FUNCTION_BLOCK FB_WriteHPTSettings
VAR_INPUT
END_VAR
VAR_OUTPUT
END_VAR
VAR
	WriteSetting	: FB_WriteSDO;
	Step			: INT := 1;
	Debug1			: BOOL;
	DebugSize2		: BYTE;
	err				: BOOL;
	errId			: UDINT;
END_VAR

CASE Step OF

1:
// Write Thermocouple Ch1 settings
WriteSetting(
	nSlaveAddr := 1011,
	nIndex := 16#8000,
	nSubIndex := 16#01,
	bExecute := TRUE,
	nValueBool := 16#01
);

Debug1 := TO_BOOL(WriteSetting.nValueBool);

IF WriteSetting.bBusy = FALSE THEN
	Step := Step +1;
END_IF

2:
WriteSetting(
	nSlaveAddr := 1011,
	nIndex := 16#8000,
	nSubIndex := 16#07,
	nValueBool := 16#01,
	bExecute := TRUE
);

IF WriteSetting.bBusy = FALSE THEN
	Step := Step +1;
END_IF

3:
WriteSetting(
	nSlaveAddr := 1011,
	nIndex := 16#8000,
	nSubIndex := 16#08,
	nValueBool := 16#01,
	bExecute := TRUE
);

IF WriteSetting.bBusy = FALSE THEN
	Step := Step +1;
END_IF

4:
WriteSetting(
	nSlaveAddr := 1011,
	nIndex := 16#8000,
	nSubIndex := 16#12,
	nValueDInt := 31451,
	bExecute := TRUE
);

IF WriteSetting.bBusy = FALSE THEN
	Step := Step +1;
END_IF

5:
WriteSetting(
	nSlaveAddr := 1011,
	nIndex := 16#8000,
	nSubIndex := 16#13,
	nValueInt := -730,
	bExecute := TRUE
);

IF WriteSetting.bBusy = FALSE THEN
	Step := Step +1;
END_IF

6:
WriteSetting(
	nSlaveAddr := 1011,
	nIndex := 16#8000,
	nSubIndex := 16#14,
	nValueInt := 4820,
	bExecute := TRUE
);

IF WriteSetting.bBusy = FALSE THEN
	Step := Step +1;
END_IF

7:
// Write Thermocouple Ch2 settings
WriteSetting(
	nSlaveAddr := 1011,
	nIndex := 16#8010,
	nSubIndex := 16#01,
	nValueBool := 16#01,
	bExecute := TRUE
);

IF WriteSetting.bBusy = FALSE THEN
	Step := Step +1;
END_IF

8:
WriteSetting(
	nSlaveAddr := 1011,
	nIndex := 16#8010,
	nSubIndex := 16#07,
	nValueBool := 16#01,
	bExecute := TRUE
);

IF WriteSetting.bBusy = FALSE THEN
	Step := Step +1;
END_IF

9:
WriteSetting(
	nSlaveAddr := 1011,
	nIndex := 16#8010,
	nSubIndex := 16#08,
	nValueBool := 16#01,
	bExecute := TRUE
);

IF WriteSetting.bBusy = FALSE THEN
	Step := Step +1;
END_IF

10:
WriteSetting(
	nSlaveAddr := 1011,
	nIndex := 16#8010,
	nSubIndex := 16#12,
	nValueDInt := 31451,
	bExecute := TRUE
);

IF WriteSetting.bBusy = FALSE THEN
	Step := Step +1;
END_IF

11:
WriteSetting(
	nSlaveAddr := 1011,
	nIndex := 16#8010,
	nSubIndex := 16#13,
	nValueInt := -730,
	bExecute := TRUE
);

IF WriteSetting.bBusy = FALSE THEN
	Step := Step +1;
END_IF

12:
WriteSetting(
	nSlaveAddr := 1011,
	nIndex := 16#8010,
	nSubIndex := 16#14,
	nValueInt := 4820,
	bExecute := TRUE,
	bError => err,
	nErrId => errid
);

(*
// Write EL5042 encoder settings to enable correct readout
WriteSetting(
	nSlaveAddr := 1010,
	nIndex := 16#8008,
	nSubIndex := 16#15,
	nValue := 26,
	bExecute := TRUE
);

WriteSetting(
	nSlaveAddr := 1010,
	nIndex := 16#8008,
	nSubIndex := 16#16,
	nValue := 0,
	bExecute := TRUE
);

WriteSetting(
	nSlaveAddr := 1010,
	nIndex := 16#8018,
	nSubIndex := 16#15,
	nValue := 26,
	bExecute := TRUE
);

WriteSetting(
	nSlaveAddr := 1010,
	nIndex := 16#8018,
	nSubIndex := 16#16,
	nValue := 0,
	bExecute := TRUE
);
*)
Step := 1;
END_CASE

END_FUNCTION_BLOCK

(* stored: Version 1.1.0.1, ProductVersion 3.1.4024.2
   POU FB_WriteHPTSettings: Id {184ad57b-2912-4b22-abd5-636de5b01f6d}, SpecialFunc None *)
